INTERFACE I_Derived EXTENDS I_Base

METHOD Derived : BOOL
VAR_INPUT
END_VAR
END_METHOD

END_INTERFACE

(* stored: Version 1.1.0.1, ProductVersion 3.1.4024.12
   Itf I_Derived: Id {c3542b46-e56a-4beb-8f31-14f9b77c89b7}
   Method Derived: Id {9e2a1c12-e644-468d-9b51-cab910afc185} *)
